SUBAPPLICATION Ventilsteuerung_Uebung_013 (* SR-Flip-Flop (Softkey) *)
  (* Standard: 61499-2 *)
  (* Version 1.0, 2023-10-23, franz *)
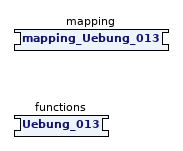
  SUBAPPS
    mapping : mapping_Uebung_013;
    functions : Uebung_013;
  END_SUBAPPS
END_SUBAPPLICATION
